// TIA Portal V17 export
// export: Created 2024-09-02T12:50:28.3458963Z, ExportSetting WithDefaults, DisplayName Totally Integrated Automation Portal, DisplayVersion V17, DisplayName TIA Portal Openness, DisplayVersion V17, DisplayName TIA Portal Version Control Interface, DisplayVersion V17, DisplayName STEP 7 Professional, DisplayVersion V17, DisplayName STEP 7 Safety, DisplayVersion V17, DisplayName WinCC Professional, DisplayVersion V17
TYPE "TypeFunction"
// stored: IsFailsafeCompliant false
   STRUCT
      Function : Array[1..348] of Struct   // Funktion / Function
         active : Bool;
         left : Bool;
         right : Bool;
         ConfigFault : Bool;
      END_STRUCT;
      Function_aktiv : Bool;   // mindestens eine Funktion aktiv / At least one function active
      Nr_Function_aktiv : Int;   // Anzahl Funktion aktiv / Number of function active
      int_Counter : Int := 1;   // Statisch Zahler / Static payer
      int_Func_Counter : Int;   // Statisch Funktionszaehler / Static Function counter
      int_Nr_Function : Int;   // Statisch Anzahl Funktionen / Static Number of functions
   END_STRUCT;
END_TYPE
